FUNCTION_BLOCK fbMultipleArmBasketMemory
VAR_INPUT
END_VAR
VAR_OUTPUT
END_VAR
VAR
END_VAR

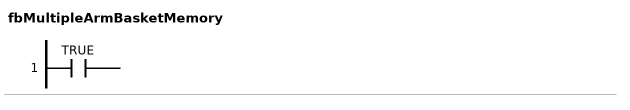
// NETWORK 1

END_FUNCTION_BLOCK

(* stored: Version 1.1.0.1, ProductVersion 3.1.4024.12
   POU fbMultipleArmBasketMemory: Id {dc7f97f8-de22-4e41-a0cd-af5b8557ba9c}, SpecialFunc None *)
